// TwinCAT 3 PLC project B_LogMessageWithArg
// ProgramVersion: 3.1.4023.0
// libraries:
//   Log4TC, * (mbc engineering GmbH)
//   Tc2_Standard, * (Beckhoff Automation GmbH)
//   Tc2_System, * (Beckhoff Automation GmbH)
//   Tc3_Module, * (Beckhoff Automation GmbH)
// project tree:
//   / MAIN.TcPOU, PlcTask.TcTTO
// (motion and I/O tree: see PLC project a_simplelogmessage)
// real-time tasks:
//   TASK PlcTask: cycle T#10ms, priority 20, ADS port 350
//   TASK PlcTask1: cycle T#10ms, priority 21, ADS port 351
//   TASK PlcTask2: cycle T#10ms, priority 22, ADS port 352

CONFIGURATION B_LogMessageWithArg
    RESOURCE PLC ON TwinCAT3
        TASK PlcTask(INTERVAL := T#10ms, PRIORITY := 20);
        PROGRAM MAIN WITH PlcTask : MAIN;
    END_RESOURCE
END_CONFIGURATION

// ---- MAIN.TcPOU
PROGRAM MAIN
VAR
	nCounter	: UINT;
	fbCountTime	: TON := (PT:=T#1S);
END_VAR

IF _TaskInfo[GETCURTASKINDEXEX()].FirstCycle THEN
	// For Remote Log4TC Server change the AMS net ID and configure a route
	PRG_TaskLog.Init('192.168.56.1.1.1');
	F_Log(E_LogLevel.eInfo, 'SPS Task gestartet.');
END_IF

fbCountTime(IN:=NOT fbCountTime.Q);
IF fbCountTime.Q THEN
	nCounter := nCounter + 1;
	F_LogA1(E_LogLevel.eInfo, 'Zähler geändert, neuer Wert {0}', nCounter);
END_IF

PRG_TaskLog.Call();

END_PROGRAM
